// TIA Portal V17 export
// export: Created 2025-03-10T12:19:28.4748584Z, ExportSetting WithDefaults, DisplayName Totally Integrated Automation Portal, DisplayVersion V17 Update 8, DisplayName TIA Portal Openness, DisplayVersion V17 Update 8, DisplayName TIA Portal Version Control Interface, DisplayVersion V17, DisplayName SINAMICS Startdrive Advanced, DisplayVersion V17 SP2, DisplayName SINAMICS Startdrive G110M, G120, G120C, G120D, G120P, G115D, DisplayVersion V17 SP2, DisplayName SINAMICS Startdrive G130, G150, S120, S150, SINAMICS MV, S210, DisplayVersion V17 SP2, DisplayName STEP 7 Professional, DisplayVersion V17 Update 8, DisplayName SINUMERIK ONE STEP 7 Toolbox, DisplayVersion V17 Update 12, DisplayName SINUMERIK 840D sl STEP 7 Toolbox, DisplayVersion V17 Update 12, DisplayName STEP 7 Safety, DisplayVersion V17 Update 6, DisplayName WinCC Advanced, DisplayVersion V17 Update 8
TYPE "UDT_Hopper Line"
// stored: IsFailsafeCompliant false
   STRUCT
      STIRRER_SPEED_ACTUAL : DInt;   // STIRRER SPEED - ACTUAL
      STIRRER_SPEED_MANUAL : DInt;   // STIRRER SPEED - MANUAL
      STIRRER_SPEED_AUTO : DInt;   // STIRRER SPEED - AUTO
      TEMP_UPPER_JACKET_ACTUAL : Real;   // TEMP UPPER JACKET - ACTUAL
      TEMP_UPPER_JACKET_MANUAL : Real;   // TEMP UPPER JACKET - MANUAL
      TEMP_UPPER_JACKET_AUTO : Real;   // TEMP UPPER JACKET - AUTO
      TEMP_LOWER_JACKET_ACTUAL : Real;   // TEMP LOWER JACKET - ACTUAL
      TEMP_LOWER_JACKET_MANUAL : Real;   // TEMP LOWER JACKET - MANUAL
      TEMP_LOWER_JACKET_AUTO : Real;   // TEMP LOWER JACKET - AUTO
      MAX_WEIGHT_ACTUAL : Real;   // MAX WEIGHT - ACTUAL
      MAX_WEIGHT_MANUAL : Real;   // MAX WEIGHT - MANUAL
      TOTAL_WEIGHT_ACTUAL : Real;   // TOTAL WEIGHT - ACTUAL
      HOPPER_WEIGHT_ACTUAL : Real;   // HOPPER WEIGHT - ACTUAL
      HOPPER_WEIGHT_MANUAL : Real;   // HOPPER WEIGHT - MANUAL
      POWDER_WEIGHT_ACTUAL : Real;   // POWDER WEIGHT - ACTUAL
      HOPPER_COVER_ACTUAL : Real;   // HOPPER COVER- ACTUAL
      HOPPER_COVER_MANUAL : Real;   // HOPPER COVER - MANUAL
      HOPPER_COVER_AUTO : Real;   // HOPPER COVER - AUTO
      FEEDING_COVER_ACTUAL : Real;   // FEEDING COVER - ACTUAL
      FEEDER_DISK_PRESSURE_ACTUAL : Real;   // FEEDER DISK PRESSURE- ACTUAL
      POWDER_FEEDER_WEIGHT_ACTUAL : Real;   // POWDER FEEDER WEIGHT ACTUAL
      TRANSFER_POWDER_SEQ_START : Bool;   // TRANSFER POWDER SEQ - START
      TRANSFER_POWDER_SEQ_STOP : Bool;   // TRANSFER POWDER SEQ - STOP
      PRESSURIZE_GAS_VALVE_START : Bool;   // PRESSURIZE GAS VALVE - START
      PRESSURIZE_GAS_VALVE_STOP : Bool;   // PRESSURIZE GAS VALVE - STOP
      RELIEVE_GAS_VALVE_START : Bool;   // RELIEVE GAS VALVE - START
      RELIEVE_GAS_VALVE_STOP : Bool;   // RELIEVE GAS VALVE - STOP
      CLEANING_AIR_VALVE_START : Bool;   // CLEANING AIR VALVE - START
      CLEANING_AIR_VALVE_STOP : Bool;   // CLEANING AIR VALVE - STOP
      LOAD_FEEDER_SEQUENCE_START : Bool;   // LOAD FEEDER SEQUENCE - START
      LOAD_FEEDER_SEQUENCE_STOP : Bool;   // LOAD FEEDER SEQUENCE - STOP
      STIRRER_STARTED : Bool;   // STIRRER - STARTED
      TEMP_UPPER_JACKET_STARTED : Bool;   // TEMP UPPER JACKET - STARTED
      TEMP_LOWER_JACKET_STARTED : Bool;   // TEMP LOWER JACKET - STARTED
      HOPPER_COVER_STARTED : Bool;   // HOPPER COVER - STARTED
   END_STRUCT;
END_TYPE
